GLOBALCONSTANTS DataPanel_MI_AI (* DataPanel Modules with medium IO density AI constants *)
  (* Standard: 61499-1; Description: Copyright (c) 2026 HR Agrartechnik GmbH *)
  (* Version 1.0, 2026-01-16, generated, HR Agrartechnik GmbH *)
  PACKAGE DataPanel::io::MI::AI;
  VAR_GLOBAL CONSTANT
    AnalogInput_1A : DataPanel::io::MI::AI::DataPanel_MI_AI_S := (Pin := 1);
    AnalogInput_1B : DataPanel::io::MI::AI::DataPanel_MI_AI_S := (Pin := 2);
    AnalogInput_2A : DataPanel::io::MI::AI::DataPanel_MI_AI_S := (Pin := 3);
    AnalogInput_2B : DataPanel::io::MI::AI::DataPanel_MI_AI_S := (Pin := 4);
    AnalogInput_3A : DataPanel::io::MI::AI::DataPanel_MI_AI_S := (Pin := 5);
    AnalogInput_3B : DataPanel::io::MI::AI::DataPanel_MI_AI_S := (Pin := 6);
    AnalogInput_4A : DataPanel::io::MI::AI::DataPanel_MI_AI_S := (Pin := 7);
    AnalogInput_4B : DataPanel::io::MI::AI::DataPanel_MI_AI_S := (Pin := 8);
    AnalogInput_5A : DataPanel::io::MI::AI::DataPanel_MI_AI_S := (Pin := 9);
    AnalogInput_5B : DataPanel::io::MI::AI::DataPanel_MI_AI_S := (Pin := 10);
    AnalogInput_6A : DataPanel::io::MI::AI::DataPanel_MI_AI_S := (Pin := 11);
    AnalogInput_6B : DataPanel::io::MI::AI::DataPanel_MI_AI_S := (Pin := 12);
    AnalogInput_7A : DataPanel::io::MI::AI::DataPanel_MI_AI_S := (Pin := 13);
    AnalogInput_7B : DataPanel::io::MI::AI::DataPanel_MI_AI_S := (Pin := 14);
    AnalogInput_8A : DataPanel::io::MI::AI::DataPanel_MI_AI_S := (Pin := 15);
    AnalogInput_8B : DataPanel::io::MI::AI::DataPanel_MI_AI_S := (Pin := 16);
    Invalid : DataPanel::io::MI::AI::DataPanel_MI_AI_S := (Pin := 255);
  END_VAR
END_GLOBALCONSTANTS
